VAR_GLOBAL
	// Einbruchbild
	L_EinbruchBild : STRING;
	// Bild der Wolke (Wetter)
	WetterBild : STRING := BildWolke;
	// Bild Licht (Im Haus)
	BildLicht : STRING := GVL_Constants.BildLicht;
END_VAR

(* stored: Version 1.1.0.1, ProductVersion 3.1.4018.5
   GVL Haus1: Id {7591fdef-56cc-4e1d-bcd8-c11f2b12c89e} *)
